KUKA KRL data list: CheckCamadaP1.dat

&ACCESS RVP
DEFDAT  CHECKCAMADAP1
;FOLD EXTERNAL DECLARATIONS;%{PE}%MKUKATPBASIS,%CEXT,%VCOMMON,%P
;FOLD BASISTECH EXT;%{PE}%MKUKATPBASIS,%CEXT,%VEXT,%P
EXT  BAS (BAS_COMMAND  :IN,REAL  :IN )
DECL INT SUCCESS
;ENDFOLD (BASISTECH EXT)
;FOLD USER EXT;%{E}%MKUKATPUSER,%CEXT,%VEXT,%P
;Make your modifications here

;ENDFOLD (USER EXT)
;ENDFOLD (EXTERNAL DECLARATIONS)
DECL BASIS_SUGG_T LAST_BASIS={POINT1[] "Topo1E21                ",POINT2[] "Topo1E21                ",CP_PARAMS[] "CPDAT3                  ",PTP_PARAMS[] "PDAT13                  ",CONT[] "C_DIS                   ",CP_VEL[] "0.15                    ",PTP_VEL[] "100                     ",SYNC_PARAMS[] "SYNCDAT                 ",SPL_NAME[] "S0                      ",A_PARAMS[] "ADAT0                   "}
DECL E6POS XAPP1PALLET1={X 1033.50830,Y 1758.07593,Z 2000.00,A -8.18113648E-08,B -9.12006202E-14,C -180.000,S 2,T 3,E1 0.0,E2 0.0,E3 0.0,E4 0.0,E5 0.0,E6 0.0}
DECL FDAT FApp1Pallet1={TOOL_NO 1,BASE_NO 0,IPO_FRAME #BASE,POINT2[] " "}
DECL PDAT PPDAT6={VEL 100.000,ACC 100.000,APO_DIST 200.000,APO_MODE #CDIS,GEAR_JERK 50.0000,EXAX_IGN 0}
DECL E6POS XP1={X 1033.50830,Y 1758.07593,Z 2000.00,A -8.18113648E-08,B -9.12006202E-14,C -180.000,S 2,T 3,E1 0.0,E2 0.0,E3 0.0,E4 0.0,E5 0.0,E6 0.0}
DECL FDAT FP1={TOOL_NO 1,BASE_NO 0,IPO_FRAME #BASE,POINT2[] " "}
DECL PDAT PPDAT1={VEL 100.000,ACC 50.0000,APO_DIST 100.000,APO_MODE #CDIS,GEAR_JERK 50.0000,EXAX_IGN 0}
DECL E6POS XP2={X 1033.50830,Y 1758.07593,Z 2000.00,A -8.18113648E-08,B -9.12006202E-14,C -180.000,S 2,T 3,E1 0.0,E2 0.0,E3 0.0,E4 0.0,E5 0.0,E6 0.0}
DECL FDAT FP2={TOOL_NO 1,BASE_NO 0,IPO_FRAME #BASE,POINT2[] " "}
DECL LDAT LCPDAT1={VEL 2.00000,ACC 100.000,APO_DIST 100.000,APO_FAC 50.0000,AXIS_VEL 100.000,AXIS_ACC 100.000,ORI_TYP #VAR,CIRC_TYP #BASE,JERK_FAC 50.0000,GEAR_JERK 50.0000,EXAX_IGN 0}
DECL E6POS XP3={X 1460.00,Y -40.0000,Z 1999.99622,A -89.2725830,B 1.71508078E-14,C 180.000,S 2,T 2,E1 0.0,E2 0.0,E3 0.0,E4 0.0,E5 0.0,E6 0.0}
DECL FDAT FP3={TOOL_NO 1,BASE_NO 0,IPO_FRAME #BASE,POINT2[] " "}
DECL PDAT PPDAT2={VEL 100.000,ACC 100.000,APO_DIST 100.000,GEAR_JERK 50.0000,EXAX_IGN 0}
DECL E6POS XP4={X -108.716446,Y -1939.39404,Z 472.006073,A -0.109658942,B 3.69518166E-15,C 180.000,S 2,T 42,E1 0.0,E2 0.0,E3 0.0,E4 0.0,E5 0.0,E6 0.0}
DECL FDAT FP4={TOOL_NO 1,BASE_NO 0,IPO_FRAME #BASE,POINT2[] " ",TQ_STATE FALSE}
DECL PDAT PPDAT3={VEL 100.000,ACC 15.0000,APO_DIST 100.000,APO_MODE #CDIS,GEAR_JERK 50.0000,EXAX_IGN 0}
DECL E6POS XP5={X -97.9360046,Y -1903.95923,Z -429.408569,A -0.452628851,B 9.79315353E-16,C 180.000,S 2,T 42,E1 0.0,E2 0.0,E3 0.0,E4 0.0,E5 0.0,E6 0.0}
DECL FDAT FP5={TOOL_NO 1,BASE_NO 0,IPO_FRAME #BASE,POINT2[] " ",TQ_STATE FALSE}
DECL LDAT LCPDAT2={VEL 2.00000,ACC 15.0000,APO_DIST 100.000,APO_FAC 50.0000,AXIS_VEL 100.000,AXIS_ACC 100.000,ORI_TYP #VAR,CIRC_TYP #BASE,JERK_FAC 50.0000,GEAR_JERK 50.0000,EXAX_IGN 0}
DECL E6POS XP6={X -97.8002243,Y -1901.23950,Z 294.298492,A -0.452342719,B -0.00529907923,C -179.878265,S 2,T 42,E1 0.0,E2 0.0,E3 0.0,E4 0.0,E5 0.0,E6 0.0}
DECL FDAT FP6={TOOL_NO 1,BASE_NO 0,IPO_FRAME #BASE,POINT2[] " ",TQ_STATE FALSE}
DECL LDAT LCPDAT3={VEL 2.00000,ACC 100.000,APO_DIST 100.000,APO_FAC 50.0000,AXIS_VEL 100.000,AXIS_ACC 100.000,ORI_TYP #VAR,CIRC_TYP #BASE,JERK_FAC 50.0000,GEAR_JERK 50.0000,EXAX_IGN 0}
DECL MODULEPARAM_T LAST_TP_PARAMS={PARAMS[] "Kuka.PointName=P7; Kuka.FrameData.base_no=0; Kuka.FrameData.tool_no=1; Kuka.FrameData.ipo_frame=#BASE; Kuka.FrameData.point2=; Kuka.isglobalpoint=False; Kuka.MoveDataPtpName=PDAT7; Kuka.MovementDataPdat.apo_mode=#CDIS; Kuka.MovementDataPdat.apo_dist=200; Kuka.MovementData.vel=0.3; Kuka.MovementData.acc=50; Kuka.MovementData.exax_ign=0; Kuka.VelocityPtp=100; Kuka.BlendingEnabled=False; Kuka.CurrentCDSetIndex=1; Kuka.MoveDataName=CPDAT4; Kuka.MovementData.apo_fac=50; Kuka.MovementData.apo_dist=500; Kuka.MovementData.axis_acc=100; Kuka.MovementData.axis_vel=100; Kuka.MovementData.circ_typ=#BASE; Kuka.MovementData.jerk_fac=50; Kuka.MovementData.ori_typ=#VAR; Kuka.VelocityPath=0.3                    "}
DECL E6POS XP7={X 1033.50830,Y 1758.07593,Z 130.000,A -8.18113648E-08,B -9.12006202E-14,C -180.000,S 2,T 3,E1 0.0,E2 0.0,E3 0.0,E4 0.0,E5 0.0,E6 0.0}
DECL FDAT FP7={TOOL_NO 1,BASE_NO 0,IPO_FRAME #BASE,POINT2[] " "}
DECL LDAT LCPDAT4={VEL 0.300000,ACC 50.0000,APO_DIST 500.000,APO_FAC 50.0000,AXIS_VEL 100.000,AXIS_ACC 100.000,ORI_TYP #VAR,CIRC_TYP #BASE,JERK_FAC 50.0000,GEAR_JERK 100.000,EXAX_IGN 0}
DECL LDAT LCPDAT5={VEL 1.00000,ACC 100.000,APO_DIST 500.000,APO_FAC 50.0000,AXIS_VEL 100.000,AXIS_ACC 100.000,ORI_TYP #VAR,CIRC_TYP #BASE,JERK_FAC 50.0000,GEAR_JERK 100.000,EXAX_IGN 0}
DECL PDAT PPDAT7={VEL 100.000,ACC 100.000,APO_DIST 200.000,APO_MODE #CDIS,GEAR_JERK 100.000,EXAX_IGN 0}
DECL E6POS XTOPOCHECKP1={X 345.924194,Y -1868.93420,Z 1749.76282,A -0.434397,B -2.78211055E-14,C 180.000,S 2,T 34,E1 0.0,E2 0.0,E3 0.0,E4 0.0,E5 0.0,E6 0.0}
DECL FDAT FTopoCheckP1={TOOL_NO 1,BASE_NO 0,IPO_FRAME #BASE,POINT2[] " ",TQ_STATE FALSE}
DECL PDAT PPDAT4={VEL 100.000,ACC 100.000,APO_DIST 100.000,APO_MODE #CDIS,GEAR_JERK 50.0000,EXAX_IGN 0}
DECL E6POS XTOPOCHECKPROG3={X 606.038757,Y 1976.47144,Z 1000.00,A 88.7955475,B 1.33370528E-13,C -180.000,S 2,T 11,E1 0.0,E2 0.0,E3 0.0,E4 0.0,E5 0.0,E6 0.0}
DECL FDAT FTopoCheckProg3={TOOL_NO 1,BASE_NO 0,IPO_FRAME #BASE,POINT2[] " ",TQ_STATE FALSE}
DECL PDAT PPDAT5={VEL 100.000,ACC 100.000,APO_DIST 100.000,APO_MODE #CDIS,GEAR_JERK 50.0000,EXAX_IGN 0}
DECL PDAT PPDAT8={VEL 100.000,ACC 100.000,APO_DIST 100.000,APO_MODE #CDIS,GEAR_JERK 50.0000,EXAX_IGN 0}
DECL E6POS XTopoCheckP2={X 829.456299,Y 1994.85071,Z 313.769348,A 88.7955475,B 1.19905670E-12,C -180.000,S 2,T 3,E1 0.0,E2 0.0,E3 0.0,E4 0.0,E5 0.0,E6 0.0}
DECL FDAT FTopoCheckP2={TOOL_NO 1,BASE_NO 0,IPO_FRAME #BASE,POINT2[] " ",TQ_STATE FALSE}
DECL PDAT PPDAT9={VEL 100.000,ACC 100.000,APO_DIST 100.000,APO_MODE #CDIS,GEAR_JERK 50.0000,EXAX_IGN 0}
DECL E6POS XTopoCheckProg4={X 606.038757,Y 1976.47144,Z 313.769379,A 88.7955475,B -1.91525927E-13,C 180.000,S 2,T 3,E1 0.0,E2 0.0,E3 0.0,E4 0.0,E5 0.0,E6 0.0}
DECL FDAT FTopoCheckProg4={TOOL_NO 1,BASE_NO 0,IPO_FRAME #BASE,POINT2[] " ",TQ_STATE FALSE}
DECL E6POS XLIMITECHECKP2={X 606.038757,Y 1976.47144,Z 313.769379,A 88.7955475,B -1.91525927E-13,C 180.000,S 2,T 3,E1 0.0,E2 0.0,E3 0.0,E4 0.0,E5 0.0,E6 0.0}
DECL FDAT FLimiteCheckP2={TOOL_NO 1,BASE_NO 0,IPO_FRAME #BASE,POINT2[] " ",TQ_STATE FALSE}
DECL PDAT PPDAT10={VEL 100.000,ACC 100.000,APO_DIST 100.000,APO_MODE #CDIS,GEAR_JERK 50.0000,EXAX_IGN 0}
DECL E6POS XLimiteCheckP1={X 606.038757,Y 1976.47144,Z 130.000,A 88.7955475,B 1.33370528E-13,C -180.000,S 2,T 11,E1 0.0,E2 0.0,E3 0.0,E4 0.0,E5 0.0,E6 0.0}
DECL FDAT FLimiteCheckP1={TOOL_NO 1,BASE_NO 0,IPO_FRAME #BASE,POINT2[] " ",TQ_STATE FALSE}
DECL LDAT LCPDAT6={VEL 2.00000,ACC 100.000,APO_DIST 100.000,APO_FAC 50.0000,AXIS_VEL 100.000,AXIS_ACC 100.000,ORI_TYP #VAR,CIRC_TYP #BASE,JERK_FAC 50.0000,GEAR_JERK 50.0000,EXAX_IGN 0}
DECL FDAT FTopo1E1={TOOL_NO 1,BASE_NO 0,IPO_FRAME #BASE,POINT2[] " ",TQ_STATE FALSE}
DECL PDAT PPDAT11={VEL 100.000,ACC 100.000,APO_DIST 100.000,APO_MODE #CDIS,GEAR_JERK 50.0000,EXAX_IGN 0}
DECL FDAT FTopo1E21={TOOL_NO 1,BASE_NO 0,IPO_FRAME #BASE,POINT2[] " ",TQ_STATE FALSE}
DECL PDAT PPDAT12={VEL 100.000,ACC 100.000,APO_DIST 100.000,APO_MODE #CDIS,GEAR_JERK 50.0000,EXAX_IGN 0}
DECL PDAT PPDAT13={VEL 100.000,ACC 100.000,APO_DIST 100.000,APO_MODE #CDIS,GEAR_JERK 50.0000,EXAX_IGN 0}
ENDDAT
